Fanuc KAREL source: kb00196.KL

PROGRAM KB00196
%STACKSIZE=65535
%PRIORITY=65535
%NOLOCKGROUP
VAR
P1 : STRING[80]
P2 : INTEGER
P3 : INTEGER
P4 : STRING[80]
BEGIN
P1='A'
P2=1
P3=1
P4='A'
VOL_SPACE(P1,P2,P3,P4)
END KB00196
